// TIA Portal V19 export
DATA_BLOCK "RandomDataGenerator_DB"   // DB8
// stored: InstanceOfName RandomDataGenerator, InstanceOfType FB
"RandomDataGenerator"
   // VAR
   //    RandInt_1 : Int;
   //    RandInt_2 : Int;
   //    RandInt_3 : Int;
   //    RandInt_4 : Int;
   //    RandInt_5 : Int;
   //    RandReal_1 : Real;
   //    RandReal_2 : Real;
   //    RandReal_3 : Real;
   //    RandReal_4 : Real;
   //    RandReal_5 : Real;
   // END_VAR
BEGIN
END_DATA_BLOCK
